FUNCTION_BLOCK SteamFlow (* Basic Function Block Type *)
  (* Standard: 61499-2 *)
  (* Version 0.0, 2011-12-21, 4DIAC-IDE, 4DIAC-Consortium *)
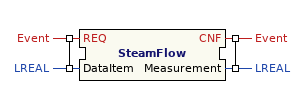
  EVENT_INPUT
    REQ WITH DataItem; (* Normal Execution Request *)
  END_EVENT
  EVENT_OUTPUT
    CNF WITH Measurement; (* Execution Confirmation *)
  END_EVENT
  VAR_INPUT
    DataItem : LREAL; (* Input event qualifier *)
  END_VAR
  VAR_OUTPUT
    Measurement : LREAL;
  END_VAR
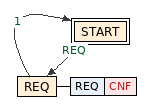
  EC_STATES
    START; (* Initial State *)
    REQ : REQ -> CNF; (* Normal execution *)
  END_STATES
  EC_TRANSITIONS
    START TO REQ := REQ;
    REQ TO START := 1;
  END_TRANSITIONS
  ALGORITHM REQ IN ST: (* Normally executed algorithm *)
Measurement:=DataItem;
  END_ALGORITHM
END_FUNCTION_BLOCK
